INTERFACE ITF_EventLog

/// sets the corresponding notification item flag raised
{attribute 'object_name' := 'SetEvent'}
METHOD SetEvent //: REFERENCE TO ST_Event
VAR_INPUT
	/// item to set
	stEvent			: ST_Event;
END_VAR
END_METHOD

END_INTERFACE

(* stored: Version 1.1.0.1
   Itf ITF_EventLog: Id {498c23bb-0d23-4478-9768-8b7efd3d3565}
   Method SetEvent: Id {c1b67bf1-5bb7-4157-a82a-7f12627e9cf8} *)
